// LS Electric XG5000 project: 동남80_1
// PLC NewPLC
// module base 0 slot 0: 입출력 모듈:XBC-DN/DP14E (DC 24V 입력 8점, 트랜지스터 출력 6점)

PROGRAM NewProgram (task: 스캔 프로그램)

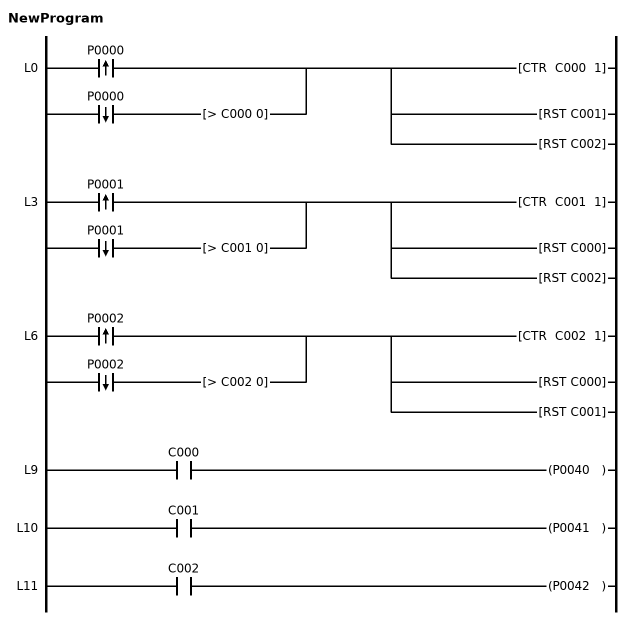
; L0
LOADP     P0000
LOADN     P0000
AND>      C000 0
OR LOAD
CTR       C000 1
RST       C001
RST       C002
; L3
LOADP     P0001
LOADN     P0001
AND>      C001 0
OR LOAD
CTR       C001 1
RST       C000
RST       C002
; L6
LOADP     P0002
LOADN     P0002
AND>      C002 0
OR LOAD
CTR       C002 1
RST       C000
RST       C001
; L9
LOAD      C000
OUT       P0040
; L10
LOAD      C001
OUT       P0041
; L11
LOAD      C002
OUT       P0042